ABB RAPID module: Module1.mod

MODULE Module1
	CONST robtarget Target_10:=[[710.302,-50.687,666.042],[0,1,0,0],[-1,0,1,0],[9E+09,9E+09,9E+09,9E+09,9E+09,9E+09]];
	VAR bool i:=FALSE;
    VAR bool j:=FALSE;
    CONST robtarget Target_20:=[[760.301980587,-50.686989693,756.042035513],[-0.000000033,1,-0.000000027,0.000000018],[-1,-1,1,0],[9E+09,9E+09,9E+09,9E+09,9E+09,9E+09]];

    PROC Path_10()

        MoveL Target_10,v1000,z100,Mano_de_Juan\WObj:=wobj0;
            WaitTime 0.2;
            SetDO ActivaMano_Juan,1;
            WaitTime 0.2;
        MoveL Target_20,v1000,z100,Mano_de_Juan\WObj:=wobj0;
            WaitTime 0.2;
            SetDO ActivaMano_Juan,0;
            WaitTime 0.2;
        MoveL Target_20,v1000,z100,Mano_de_Juan\WObj:=wobj0;
            WaitTime 0.2;
            SetDO ActivaMano_Juan,1;
            WaitTime 0.2;
        MoveL Target_10,v1000,z100,Mano_de_Juan\WObj:=wobj0;
            WaitTime 0.2;
            SetDO ActivaMano_Juan,0;
            WaitTime 0.2;
            j:=TRUE;

	ENDPROC





    PROC main()

    IF i=FALSE THEN
        SetDO Cinta_on,0;
        WaitTime 1;
        SetDO Cinta_on,1;
        i:=TRUE;
    ENDIF

    IF Sensor_cinta = 1 THEN
        WaitTime 1;
        Path_10;

    IF j=TRUE AND Sensor_cinta = 1 THEN
        SetDO Montaje_fin,1;
        j:=FALSE;
    ELSE
        WaitTime 1;
        SetDO Montaje_fin,0;
    ENDIF


    ENDPROC

ENDMODULE
